// TIA Portal V20 export
TYPE "LER_typeCommunicationBRCVConfiguration"
// stored: Access Published
   STRUCT
      connectionId : CONN_PRG := 16#0;
      rid { ExternalAccessible := 'False'; ExternalVisible := 'False'; ExternalWritable := 'False'} : CONN_R_ID := 16#0;
   END_STRUCT;
END_TYPE
